{region '#Template'}
	{attribute 'Version' := '1.0.0.0'}
	{attribute 'Tags' := '"LCID": "1031", "Text": "DUT, Operation mode, Universal, 3Step"'}
	{attribute 'Tags' := '"LCID": "1033", "Text": "DUT, Operation mode, Universal, 3Step"'}
	{attribute 'Description' := '"LCID": "1031", "Text": "Betriebsart 3 3Step"'}
	{attribute 'Description' := '"LCID": "1033", "Text": "Operating mode 3 steps"'}
{endregion}

{attribute qualified_only}
TYPE E_BA_3Step :
(
	eOff			:= 1,
	eStep1			:= 2,
	eStep2			:= 3,
	eStep3			:= 4
	
) UDINT;
END_TYPE

(* stored: Version 1.1.0.1, ProductVersion 3.1.4024.9
   DUT E_BA_3Step: Id {43f6ce31-18ce-4b1c-a674-90867ccac892} *)
